FUNCTION_BLOCK FB_Controlbox
VAR_INPUT
	bRealControlBox: BOOL;
END_VAR
VAR_OUTPUT
END_VAR
VAR
	fbJoystickScaling : FB_JoystickNorm;
	fbRealControlBox : FB_RealControlBox;
	fbVirtualControlbox : FB_VirtualControlBox;
	fbSelectedControlBox : I_ControlBox;
END_VAR


fbJoystickScaling( fRawInput := task1.fJoystickX, fOutput => task1.fJoyXNormalized);
fbJoystickScaling( fRawInput := task1.fJoystickY, fOutput => task1.fJoyYNormalized);

IF bRealControlBox THEN
	fbSelectedControlBox := fbRealControlBox;
ELSE
	fbSelectedControlBox := fbVirtualControlBox;
END_IF

END_FUNCTION_BLOCK

(* stored: Version 1.1.0.1, ProductVersion 3.1.4024.12
   POU FB_Controlbox: Id {2cd6bccb-390e-458d-b579-143a077dcf5b}, SpecialFunc None *)
